TYPE ST_EP3751 :
	STRUCT
		// Unit in 1G
		ACC_X : REAL;
		ACC_Y : REAL;
		ACC_Z : REAL;
		// °/s
		Gyro_X : REAL;
		Gyro_Y : REAL;
		Gyro_Z : REAL;
	END_STRUCT
END_TYPE

(* stored: Version 1.1.0.1
   DUT ST_EP3751: Id {82ccaf5b-2a81-4b06-b0bf-8b34cac27aab} *)
